// TIA Portal V16 export
// export: Created 2023-08-28T09:37:56.2706874Z, ExportSetting WithDefaults, DisplayName Totally Integrated Automation Portal, DisplayVersion V16 Update 6, DisplayName TIA Portal Version Control Interface, DisplayVersion V16 Update 2, DisplayName TIA Portal Openness, DisplayVersion V16 Update 6, DisplayName STEP 7 Professional, DisplayVersion V16 Update 6, DisplayName STEP 7 Safety, DisplayVersion V16, DisplayName WinCC Advanced, DisplayVersion V16 Update 6
TYPE "typeModbusCommLoad"
// stored: IsFailsafeCompliant false
   STRUCT
      done : Bool := FALSE;   // Boolean indicating completion without error
      error : Bool := FALSE;   // Boolean indicating completion with error
      status : Word := W#16#0;   // Status or error code of the completed operation
      errorStatus : Word := W#16#0;   // Error code of the faulty operation
   END_STRUCT;
END_TYPE
